FUNCTION_BLOCK FB_LiftControlEmulation
VAR_INPUT	
	Config					: ST_CFG_TransferUnitEmulation; // emulation config	
	DriveRun_Lift			: BOOL;
END_VAR

VAR_OUTPUT
	Lift_Pos_Down			: BOOL;
	Lift_Pos_Up				: BOOL;
END_VAR

VAR
	ActualPosition			: INT;
	CountPositive			: BOOL;
END_VAR


// When lift is moving
IF DriveRun_Lift THEN
	IF CountPositive THEN
		IF ActualPosition < Config.Position_Max_Up THEN
			ActualPosition := ActualPosition + 1;
		ELSE
			CountPositive := FALSE;
		END_IF;	
	ELSE
		IF ActualPosition > Config.Position_Max_Down THEN
			ActualPosition := ActualPosition - 1;
		ELSE
			CountPositive := TRUE;
		END_IF;					
	END_IF
END_IF

// Update positions
IF ActualPosition = Config.Position_Down AND NOT CountPositive THEN
	 Lift_Pos_Down := TRUE;
ELSIF ActualPosition = Config.Position_Up AND CountPositive THEN
	 Lift_Pos_Up := TRUE;
ELSE
	Lift_Pos_Down := FALSE;
	Lift_Pos_Up := FALSE;
END_IF

END_FUNCTION_BLOCK

(* stored: Version 1.1.0.1, ProductVersion 3.1.4024.9
   POU FB_LiftControlEmulation: Id {122dee98-82f6-4eb7-ad42-4d8d8f66a756}, SpecialFunc None *)
